INTERFACE I_LimSwStatusShareData

PROPERTY HomeBusy : BOOL
GET
END_GET
END_PROPERTY

PROPERTY LimBackward : BOOL
SET
END_SET
END_PROPERTY

PROPERTY LimForward : BOOL
SET
END_SET
END_PROPERTY

PROPERTY LimHome : BOOL
SET
END_SET
END_PROPERTY

PROPERTY MoveBusy : BOOL
GET
END_GET
END_PROPERTY

PROPERTY NegativeDirection : BOOL
GET
END_GET
END_PROPERTY

PROPERTY NewMoveReq : BOOL
GET
END_GET
END_PROPERTY

PROPERTY PositiveDirection : BOOL
GET
END_GET
END_PROPERTY

PROPERTY ResetDone : BOOL
GET
END_GET
SET
END_SET
END_PROPERTY

END_INTERFACE

(* stored: Version 1.1.0.1
   Itf I_LimSwStatusShareData: Id {05293a1e-386a-46e0-b219-a39c6e520011}
   Property HomeBusy: Id {2382ab9e-e464-498b-b3d1-3eb574860f78}
   Get Get: Id {35889636-b658-4fba-89f2-a1033924d466}
   Property LimBackward: Id {be547acb-e1fd-4050-bb2d-6f025603040d}
   Set Set: Id {1064053d-7051-418d-af4e-8ef6837c518f}
   Property LimForward: Id {507a6415-3928-42e3-8134-3e476dbbb9d5}
   Set Set: Id {6976668a-3343-4e7d-8696-f0561798ac20}
   Property LimHome: Id {7438c6e7-800b-414c-9ad6-226a2391d055}
   Set Set: Id {76272b5c-968c-401a-a649-70372123cf48}
   Property MoveBusy: Id {5e0e073b-50c5-4948-be6f-702b298fdd9b}
   Get Get: Id {f6af31e0-cb12-4de7-b30f-e64dd9ed7440}
   Property NegativeDirection: Id {9dde2d2c-6ea8-4c4f-9a29-430cb504c6a3}
   Get Get: Id {304943df-a34e-4d56-8af4-18e58cdebd37}
   Property NewMoveReq: Id {470d22ec-d499-457f-bd91-c8f2969f0877}
   Get Get: Id {99c62cdc-4799-4413-bfd3-3fdf623fa6bb}
   Property PositiveDirection: Id {b4b9bcd8-0d26-4798-b88f-a394bea26cbf}
   Get Get: Id {cc5f8abd-898d-42b9-9407-3ac75b0da583}
   Property ResetDone: Id {f7b4446b-64dc-419d-81f1-3b9e4c9e3169}
   Get Get: Id {1753b70e-ceab-416b-a694-57df3291d784}
   Set Set: Id {3c943093-deb8-48b9-900a-7bf40f233716} *)
